// Mitsubishi GX Works2 project: 240423_신입동작우선회로   PLC: Q03UDV

PROGRAM MAIN
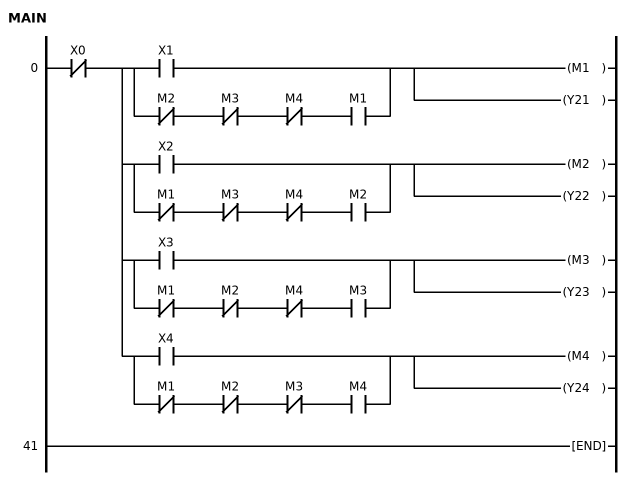
0     LDI     X0
      MPS
      LD      X1
      LDI     M2
      ANI     M3
      ANI     M4
      AND     M1
      ORB
      ANB
      OUT     M1
      OUT     Y21
      MRD
      LD      X2
      LDI     M1
      ANI     M3
      ANI     M4
      AND     M2
      ORB
      ANB
      OUT     M2
      OUT     Y22
      MRD
      LD      X3
      LDI     M1
      ANI     M2
      ANI     M4
      AND     M3
      ORB
      ANB
      OUT     M3
      OUT     Y23
      MPP
      LD      X4
      LDI     M1
      ANI     M2
      ANI     M3
      AND     M4
      ORB
      ANB
      OUT     M4
      OUT     Y24
41    END
END_PROGRAM
